// TwinCAT 3 PLC project PLC
// ProgramVersion: 3.1.4024.0
// libraries:
//   Tc2_Standard, * (Beckhoff Automation GmbH)
//   Tc2_System, * (Beckhoff Automation GmbH)
//   Tc3_Module, * (Beckhoff Automation GmbH)
// project tree:
//   / PlcTask.TcTTO
//   POUs/ MAIN.TcPOU, RampControlCycles.TcPOU, RampControlTimers.TcPOU
// real-time tasks:
//   TASK PlcTask: cycle T#10ms, priority 20, ADS port 350

CONFIGURATION PLC
    RESOURCE PLC ON TwinCAT3
        TASK PlcTask(INTERVAL := T#10ms, PRIORITY := 20);
        PROGRAM MAIN WITH PlcTask : MAIN;
    END_RESOURCE
END_CONFIGURATION

// ---- POUs/MAIN.TcPOU
PROGRAM MAIN
VAR
	RampControlCycles	:	RampControlCycles;
	RampControlTime		:	RampControlTimers;
	StartPb				: 	BOOL;
	StopPb				: 	BOOL;
END_VAR

RampControlCycles(Start:= StartPb,
			Stop := StopPb,
			RampUpTime := 15,
			ContDutyTime := 20,
			RampDownTime := 5,
			RampMinVal := 10,
			RampMaxVal := 100,
			PlcCycleTimeMs := 10);
			
			
RampControlTime(Start:= StartPb,
			Stop := StopPb,
			RampUpTime := 7,
			ContDutyTime := 10,
			RampDownTime := 5,
			RampMinVal := 5,
			RampMaxVal := 70,
			PlcCycleTimeMs := 10);

END_PROGRAM

// ---- POUs/RampControlCycles.TcPOU
FUNCTION_BLOCK RampControlCycles
VAR_INPUT
	Start					:	BOOL;
	Stop					:	BOOL;
	RampUpTime				:	UINT;				// ramp up time in seconds
	ContDutyTime			:	UINT;				// continous duty time in seconds
	RampDownTime			:	UINT;				// ramp down time in seconds
	RampMinVal				:	REAL;				// output min value
	RampMaxVal				:	REAL;				// output max value
	PlcCycleTimeMs			:	UINT;				// PLC cycle in miliseconds
END_VAR
VAR_OUTPUT
	Out						:	REAL;
	ErrorConfig				:	BOOL;
END_VAR
VAR
	rtStart					:	R_TRIG;
	rtStop					:	R_TRIG;
	SeqStep					:	(IDLE, INIT, RAMP_UP, CONTINOUS_DUTY, RAMP_DOWN);
	RampUpPoints			: 	UINT;
	RampDownPoints			: 	UINT;
	ContDutyPoints			:	UINT;
	
	RampUpValRes			:	REAL;
	RampDownValRes			:	REAL;
	RampUpCycles			:	UINT;
	RampDownCycles			:	UINT;		
	ContDutyCycles			:	UINT;
	
	InitBit					:	BOOL:=TRUE;
END_VAR

(*
This FB generates output signal ramps including three areas:
- up ramp (in seconds)
- continous duty (in seconds)
- down ramp (in seconds)

Start cycle with <Start> pulse.
The output signal can be stopped with <Stop> pulse during ramp up and cont. duty cycle. 
It ramps down in that case to avoid immediate stop (any demage of the controlled device).  
*)

IF InitBit THEN
	// check input parameters for unvalid values
	IF PlcCycleTimeMs=0 OR RampUpTime=0 OR RampDownTime=0 THEN
		ErrorConfig := TRUE;
	ELSE;
		ErrorConfig := FALSE;
	
		(*init calculations*)
		// number of cycle points during ramp up 
		RampUpPoints 	:= TO_UINT(TO_REAL(RampUpTime) / (TO_REAL(PlcCycleTimeMs) / 1000.0));
		// output value resolution for each cycle during ramp up
		RampUpValRes	:= (RampMaxVal - RampMinVal) / TO_REAL(RampUpPoints);
		
		// number of cycle points during continous duty
		ContDutyPoints := TO_UINT(TO_REAL(ContDutyTime) / (TO_REAL(PlcCycleTimeMs) / 1000.0));
		
		// number of cycle points during ramp down
		RampDownPoints	:= TO_UINT(TO_REAL(RampDownTime) / (TO_REAL(PlcCycleTimeMs) / 1000.0));
		// output value resolution for each cycle during ramp down
		RampDownValRes	:= (RampMaxVal - RampMinVal) / TO_REAL(RampDownPoints);
	END_IF
	
	InitBit			:= FALSE;
END_IF

// detect pushbuttons action
rtStart(CLK:=Start);
rtStop(CLK:=Stop);

IF rtStart.Q AND SeqStep=IDLE AND NOT ErrorConfig THEN
	SeqStep := INIT;
END_IF

IF rtStop.Q AND (SeqStep=CONTINOUS_DUTY OR SeqStep=RAMP_UP) THEN
	SeqStep := RAMP_DOWN;
END_IF


CASE SeqStep OF
	IDLE:
		;
	INIT:
		Out				:= RampMinVal;
		RampUpCycles 	:= 0;
		ContDutyCycles	:= 0;
		RampDownCycles	:= 0;
		SeqStep			:= RAMP_UP;
		
	RAMP_UP:
		Out := Out + RampUpValRes;
		RampUpCycles := RampUpCycles+1;
		IF RampUpCycles > RampUpPoints THEN SeqStep := CONTINOUS_DUTY; END_IF
		
	CONTINOUS_DUTY:
		ContDutyCycles := ContDutyCycles+1;
		IF ContDutyCycles > ContDutyPoints THEN SeqStep := RAMP_DOWN; END_IF
		
	RAMP_DOWN:
		IF (Out - RampDownValRes) > RampMinVal THEN
			Out := Out - RampDownValRes;
		ELSE
			Out := RampMinVal;
		END_IF
		
		RampDownCycles := RampDownCycles+1;
		IF RampDownCycles > RampDownPoints THEN SeqStep := IDLE; END_IF
END_CASE

END_FUNCTION_BLOCK

// ---- POUs/RampControlTimers.TcPOU
FUNCTION_BLOCK RampControlTimers
VAR_INPUT
	Start					:	BOOL;
	Stop					:	BOOL;
	RampUpTime				:	UINT;			// ramp up time in seconds
	ContDutyTime			:	UINT;			// continous duty time in seconds
	RampDownTime			:	UINT;			// ramp down time in seconds
	RampMinVal				:	REAL;			// output min value
	RampMaxVal				:	REAL;			// output max value
	PlcCycleTimeMs			:	UINT;			// PLC cycle in miliseconds
END_VAR
VAR_OUTPUT
	Out						:	REAL;
	ErrorConfig				:	BOOL;
END_VAR
VAR
	rtStart					:	R_TRIG;
	rtStop					:	R_TRIG;
	SeqStep					:	(IDLE, INIT, RAMP_UP, CONTINOUS_DUTY, RAMP_DOWN);
	
	RampUpValRes			:	REAL;
	RampDownValRes			:	REAL;	
	
	InitBit					:	BOOL:=TRUE;
	tonRampUp				:	TON;
	tonContDuty				:	TON;
	tonRampDown				:	TON;
END_VAR

(*
This FB generates output signal ramps including three areas:
- up ramp (in seconds)
- continous duty (in seconds)
- down ramp (in seconds)

Start cycle with <Start> pulse.
The output signal can be stopped with <Stop> pulse during ramp up and cont. duty cycle. 
It ramps down in that case to avoid immediate stop (any demage of the controlled device).  
*)

IF InitBit THEN
	// check input parameters for unvalid values
	IF PlcCycleTimeMs=0 OR RampUpTime=0 OR RampDownTime=0 THEN
		ErrorConfig := TRUE;
	ELSE;
		ErrorConfig := FALSE;
		(*init calculations*)
		// output value resolution for each cycle during ramp up
		RampUpValRes := (RampMaxVal - RampMinVal) / ((TO_REAL(RampUpTime) / (TO_REAL(PlcCycleTimeMs) / 1000.0)));
		// output value resolution for each cycle during ramp down
		RampDownValRes := (RampMaxVal - RampMinVal) / ((TO_REAL(RampDownTime) / (TO_REAL(PlcCycleTimeMs) / 1000.0)));
	END_IF;
	InitBit			:= FALSE;
END_IF

// detect pushbuttons action
rtStart(CLK:=Start);
rtStop(CLK:=Stop);

IF rtStart.Q AND SeqStep=IDLE AND NOT ErrorConfig THEN
	SeqStep := INIT;
END_IF

IF rtStop.Q AND (SeqStep=CONTINOUS_DUTY OR SeqStep=RAMP_UP) THEN
	SeqStep := RAMP_DOWN;
END_IF


CASE SeqStep OF
	IDLE:
		;
	INIT:
		Out				:= RampMinVal;
		tonRampUp.IN	:= FALSE;
		tonContDuty.IN	:= FALSE;
		tonRampDown.IN	:= FALSE;
		tonRampUp.PT	:= UINT_TO_TIME(RampUpTime * 1000);
		tonContDuty.PT	:= UINT_TO_TIME(ContDutyTime * 1000);
		tonRampDown.PT	:= UINT_TO_TIME(RampDownTime * 1000);
		
		SeqStep			:= RAMP_UP;
		
	RAMP_UP:
		tonRampUp.IN:= TRUE;
		Out := Out + RampUpValRes;
		IF tonRampUp.Q THEN 
			SeqStep 		:= CONTINOUS_DUTY; 
			tonRampUp.IN 	:= FALSE;
		END_IF
		
	CONTINOUS_DUTY:
		tonContDuty.IN := TRUE;
		IF tonContDuty.Q THEN
			SeqStep 		:= RAMP_DOWN;
			tonContDuty.IN 	:= FALSE;
		END_IF
		
	RAMP_DOWN:
		IF (Out - RampDownValRes) > RampMinVal THEN
			Out := Out - RampDownValRes;
		ELSE
			Out := RampMinVal;
		END_IF
		
		tonRampDown.IN	:= TRUE;
		IF tonRampDown.Q THEN
			SeqStep 		:= IDLE;
			tonRampDown.In 	:= FALSE;
		END_IF
END_CASE

tonRampUp();
tonContDuty();
tonRampDown();

END_FUNCTION_BLOCK
